{attribute addProperty BoxType "AT2040-0250-0023"}
{attribute addProperty Id "A_0106_AT2026_5250_0019_AT2026_5250AT2026_3DCFC8D064080"}
{attribute addProperty CRC "4045326406"}
{attribute addProperty SizeInBites "640"}
{attribute addProperty SizeInBytes "80"}
TYPE A_0038_AT2040_0250_0023_F11EC846 EXTENDS AT2040_9506A482 :
STRUCT
	{attribute addProperty Name "A_0106_AT2026_5250_0019_AT2026_5250"}
	A_0106_AT2026_5250_0019_AT2026_5250 : AT2026_3DCFC8D0;
END_STRUCT
END_TYPE

(* stored: Version 1.2.0.0, ProductVersion 3.1.4024.9
   DUT A_0038_AT2040_0250_0023_F11EC846: Id {a1b582e6-60a5-46ea-9324-a97cb33dc79a} *)
